PROGRAM MAIN
VAR
END_VAR

END_PROGRAM

(* stored: Version 1.1.0.1
   POU MAIN: Id {d4204e6c-b7e5-4d21-91c3-5c2c721304dd} *)
